Fanuc TP program (LS listing): T1_GRIP_COND.LS

/PROG  T1_GRIP_COND	  Cond
/ATTR
OWNER		= MNEDITOR;
COMMENT		= "monitor";
PROG_SIZE	= 172;
CREATE		= DATE 22-12-28  TIME 21:19:46;
MODIFIED	= DATE 25-07-17  TIME 09:31:30;
FILE_NAME	= ;
VERSION		= 0;
LINE_COUNT	= 1;
MEMORY_SIZE	= 548;
PROTECT		= READ_WRITE;
TCD:  STACK_SIZE	= 0,
      TASK_PRIORITY	= 50,
      TIME_SLICE	= 0,
      BUSY_LAMP_OFF	= 0,
      ABORT_REQUEST	= 0,
      PAUSE_REQUEST	= 0;
DEFAULT_GROUP	= *,*,*,*,*;
CONTROL_CODE	= 00000000 00000000;
/MN
   1:  WHEN RI[3:ON :T1 opened]=ON OR RI[4:OFF:T1 closed]=ON,CALL T1_DET_LOST ;
/POS
/END
